{attribute 'linkalways'} 
{attribute 'no_explicit_call' := 'This FB is a CLASS and must be accessed using methods or properties'}
{attribute 'enable_dynamic_creation'}
FUNCTION_BLOCK _ETcVnBarcodeSearchDirection EXTENDS EnumDatatypeBase
VAR
	localData : ETcVnBarcodeSearchDirection;
	activeData : REFERENCE TO ETcVnBarcodeSearchDirection;
	enumBaseDatatype : _UDINT(localData);
END_VAR

METHOD PRIVATE AddLocalEnumeration
VAR_INPUT
	Enumeration : T_MAXSTRING;
	Value : ETcVnBarcodeSearchDirection;
END_VAR
AddEnumeration(Enumeration, Value);
END_METHOD

PROPERTY PUBLIC Address : PVOID
GET
Address := ADR(activeData);
END_GET
END_PROPERTY

METHOD PUBLIC ClearReference
VAR_INPUT
END_VAR
activeData REF= localData;
SetBaseDatatypeReference();
END_METHOD

METHOD PUBLIC Clone : I_Datatype
VAR
    pClone : POINTER TO _ETcVnBarcodeSearchDirection;
END_VAR
pClone := __NEW(_ETcVnBarcodeSearchDirection(InitialValue := Value));
Clone := pClone^;
END_METHOD

METHOD FB_init : BOOL
VAR_INPUT
	bInitRetains : BOOL; // if TRUE, the retain variables are initialized (warm start / cold start)
	bInCopyCode : BOOL;  // if TRUE, the instance afterwards gets moved into the copy code (online change)
	InitialValue : ETcVnBarcodeSearchDirection;
END_VAR
localData := InitialValue;
AddBaseDatatype(enumBaseDatatype);
ClearReference();

AddLocalEnumeration('TCVN_BSD_ANY', ETcVnBarcodeSearchDirection.TCVN_BSD_ANY);
AddLocalEnumeration('TCVN_BSD_HORIZONTAL', ETcVnBarcodeSearchDirection.TCVN_BSD_HORIZONTAL);
AddLocalEnumeration('TCVN_BSD_VERTICAL', ETcVnBarcodeSearchDirection.TCVN_BSD_VERTICAL);
END_METHOD

PROPERTY PUBLIC Identifier : T_MAXSTRING
GET
Identifier := 'ETcVnBarcodeSearchDirection';
END_GET
END_PROPERTY

METHOD IsEnumeratorValueEqual : BOOL
VAR_INPUT
	Enumerator : I_KeyValueForwardEnumerator;
END_VAR
VAR
	storedValue : ETcVnBarcodeSearchDirection;
END_VAR
IF NOT Enumerator.TryGet(storedValue) THEN
	RETURN;
END_IF

IsEnumeratorValueEqual := storedValue = activeData;
END_METHOD

METHOD PUBLIC MakeReferenceTo
VAR_INPUT
	ReferenceTarget : REFERENCE TO ETcVnBarcodeSearchDirection;
END_VAR
activeData REF= ReferenceTarget;
SetBaseDatatypeReference();
END_METHOD

METHOD PROTECTED SetBaseDatatypeReference
VAR_INPUT
END_VAR
enumBaseDatatype.MakeReferenceTo(activeData);
END_METHOD

PROPERTY PUBLIC Size : UDINT
GET
Size := SIZEOF(activeData);
END_GET
END_PROPERTY

METHOD TryMakeReferenceTo : BOOL
VAR_INPUT
	Target : I_Datatype;
END_VAR
VAR
	targetAsEnum : I_EnumDatatype;
	pTargetData : POINTER TO ETcVnBarcodeSearchDirection;
END_VAR
IF NOT Target.TryResolveAsEnumDatatype(targetAsEnum) THEN
	RETURN;
END_IF

IF targetAsEnum.Identifier <> Identifier THEN
	RETURN;
END_IF

pTargetData := Target.Address;
activeData REF= pTargetData^;
SetBaseDatatypeReference();
TryMakeReferenceTo := TRUE;
END_METHOD

PROPERTY PUBLIC Value : ETcVnBarcodeSearchDirection
GET
Value := activeData;
END_GET
SET
activeData := Value;
END_SET
END_PROPERTY

END_FUNCTION_BLOCK

(* stored: Version 1.1.0.1
   POU _ETcVnBarcodeSearchDirection: Id {7949b088-9098-0927-1894-fa02da68710e}, SpecialFunc None
   Folder Constructor: Id {643739f9-fd7e-0f0f-228c-aaadf7a277d8}
   Folder Private: Id {f3928649-b46a-07d9-03d2-f7a28205b1e5}
   Folder Protected: Id {b18f1a73-136d-0aa0-15c2-d210a1f2f4ca}
   Method AddLocalEnumeration: Id {0437d9ce-3d70-00cf-1967-8a76dfc953cb}
   Property Address: Id {3cbd8f42-5c96-0e78-3705-daf04cc6e77f}
   Get Get: Id {728b3f11-02b4-0789-2ee0-55f72622b377}
   Method ClearReference: Id {8e326e38-d299-0882-113b-c7813798ab8e}
   Method Clone: Id {63905d34-985f-07bb-1e35-7d03d1609b6c}
   Method FB_init: Id {21fc58ed-62b2-0972-1026-c18d1e79fbd5}
   Property Identifier: Id {19517c6f-696d-0b37-2919-b26caf11a6c2}
   Get Get: Id {e1765b43-9705-07ac-13fe-09fd9bfdbf11}
   Method IsEnumeratorValueEqual: Id {773c87f6-d75d-07b0-0c88-b78cda047b81}
   Method MakeReferenceTo: Id {6482af37-678e-0887-0a9d-d86bfdd1665c}
   Method SetBaseDatatypeReference: Id {ceedcc1b-8c34-0eeb-3a1f-f8f126a571df}
   Property Size: Id {80344139-7580-0c85-08c1-939ab5bcc4e6}
   Get Get: Id {508712da-e934-0bc8-0107-38d018455eb3}
   Method TryMakeReferenceTo: Id {2dd4bcfc-8e6b-005e-28f9-f7fd9e2801fc}
   Property Value: Id {297b5bb8-4e1a-02cc-342a-d3a0b024bddb}
   Get Get: Id {9c5ffb4d-1a1e-085c-0665-b28659828410}
   Set Set: Id {379b465e-e299-0a0c-2735-cc7e0a3afc1f} *)
